Omron CX-Programmer project NewProject (CX-Programmer 9.75)

# PLC NewPLC1: CP1E E20

## Program NewProgram1 (cyclic task 0)

### Section Section1

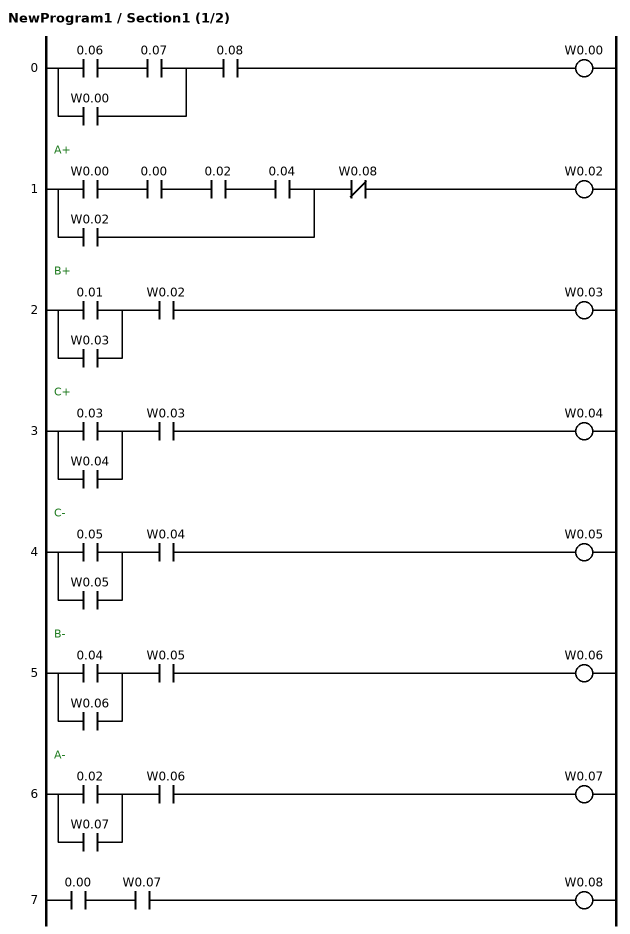
; rung 0
LD 0.06
AND 0.07
OR W0.00
AND 0.08
OUT W0.00
; rung 1: A+
LD W0.00
AND 0.00
AND 0.02
AND 0.04
OR W0.02
ANDNOT W0.08
OUT W0.02
; rung 2: B+
LD 0.01
OR W0.03
AND W0.02
OUT W0.03
; rung 3: C+
LD 0.03
OR W0.04
AND W0.03
OUT W0.04
; rung 4: C-
LD 0.05
OR W0.05
AND W0.04
OUT W0.05
; rung 5: B-
LD 0.04
OR W0.06
AND W0.05
OUT W0.06
; rung 6: A-
LD 0.02
OR W0.07
AND W0.06
OUT W0.07
; rung 7
LD 0.00
AND W0.07
OUT W0.08

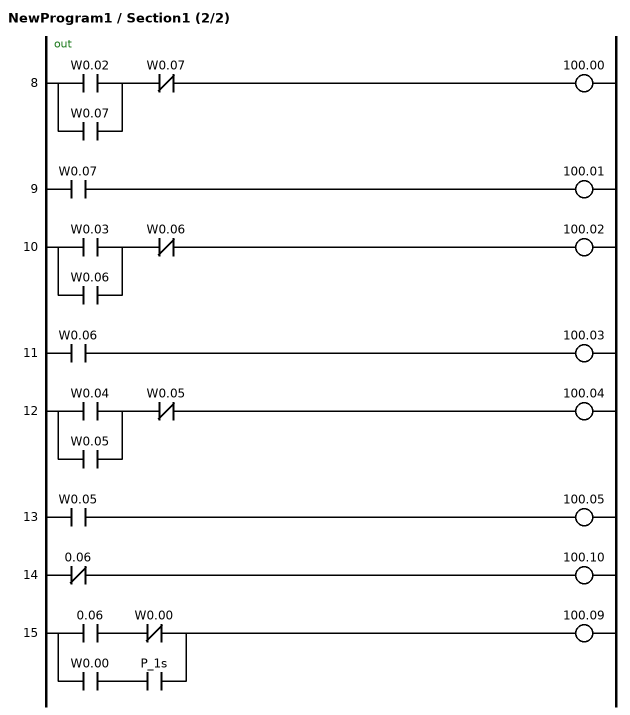
; rung 8: out
LD W0.02
OR W0.07
ANDNOT W0.07
OUT 100.00
; rung 9
LD W0.07
OUT 100.01
; rung 10
LD W0.03
OR W0.06
ANDNOT W0.06
OUT 100.02
; rung 11
LD W0.06
OUT 100.03
; rung 12
LD W0.04
OR W0.05
ANDNOT W0.05
OUT 100.04
; rung 13
LD W0.05
OUT 100.05
; rung 14
LDNOT 0.06
OUT 100.10
; rung 15
LD 0.06
ANDNOT W0.00
LD W0.00
AND P_1s
ORLD
OUT 100.09

### Section END
; rung 0
END(001)